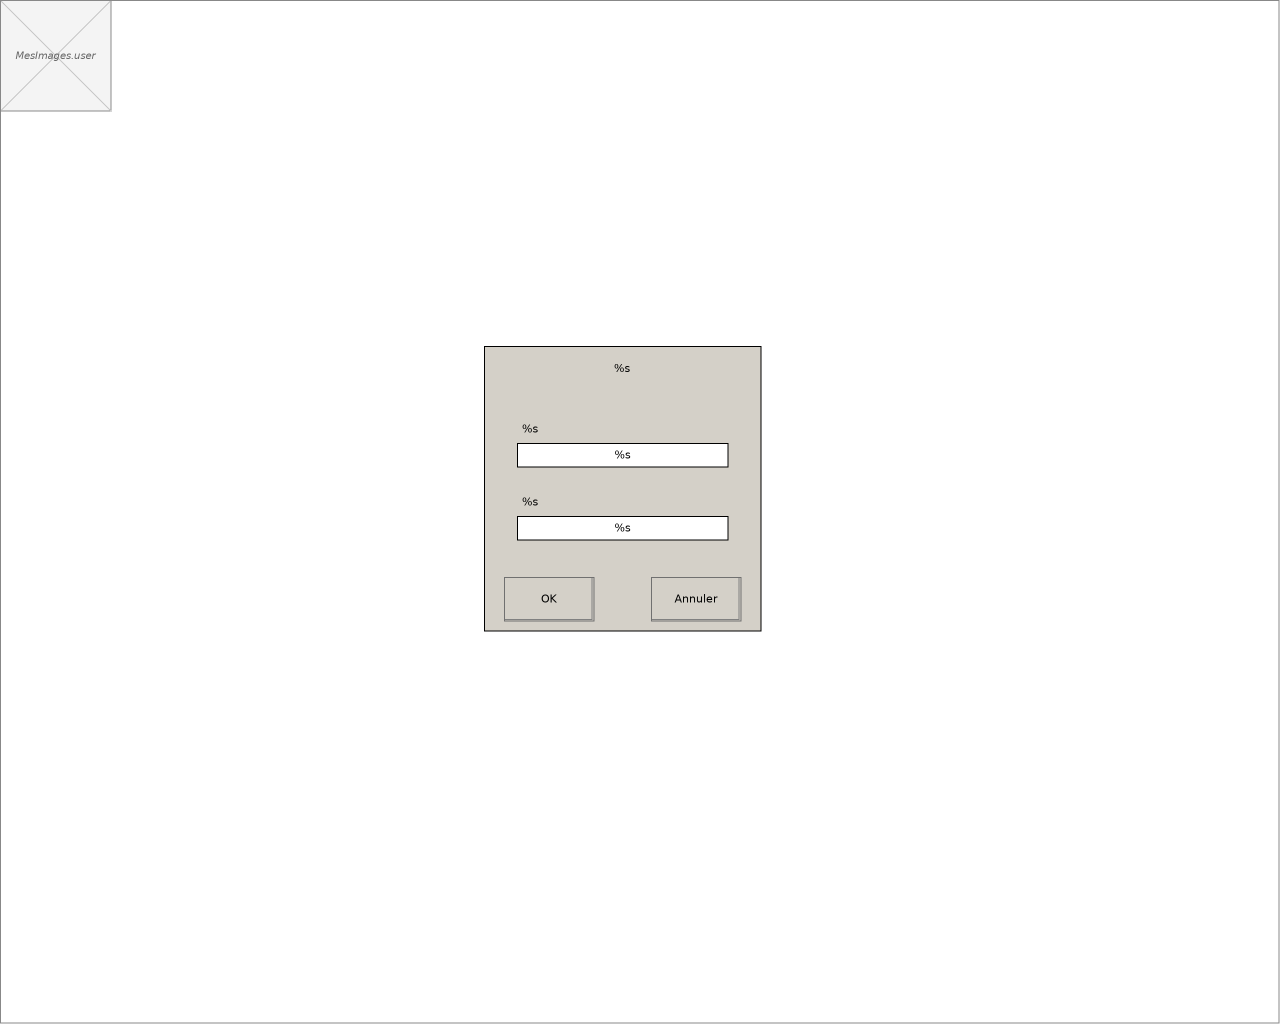
VISUALIZATION UTIL_LOG  // 1280x1024
    Image (0,0 111x111), image: MesImages.user
    RoundedRectangle (484,346 277x285)
    Textfield (503,356 238x25), "%s", text list: 'TextList_Users_Menu', text index: 4
    Button (504,577 90x44), "OK"
        toggle PRG_USER.DD_LOG
        OnMouseClick: change screen: UTIL_MENU
    Button (651,577 90x44), "Annuler"
        OnMouseClick: change screen: UTIL_MENU
    Rectangle (517,443 211x24), "%s", text variable: PRG_USER.LOG_TEMP
        OnMouseClick: write the text variable via InputWithLimits
    Rectangle (517,516 211x24), "%s", text variable: PRG_USER.PASS_TEMP_DISPLAY
        OnMouseClick: write PRG_USER.PASS_TEMP via InputWithLimits, password
    Textfield (519,419 126x20), "%s", text list: 'TextList_Users_Menu', text index: 5
    Textfield (519,492 126x20), "%s", text list: 'TextList_Users_Menu', text index: 6
END_VISUALIZATION

(* stored: Version 1.1.0.1, ProductVersion 3.1.4024.10
   Visu UTIL_LOG: Id {3afbe80b-2fa3-4a65-8888-1c0f55e02e36} *)
